// TIA Portal V18 export
// export: Created 2026-06-08T16:52:55.5874896Z, ExportSetting WithDefaults, DisplayName Totally Integrated Automation Portal, DisplayVersion V18, DisplayName TIA Portal Openness, DisplayVersion V18, DisplayName TIA Portal Version Control Interface, DisplayVersion V18, DisplayName STEP 7 Professional, DisplayVersion V18, DisplayName STEP 7 Safety, DisplayVersion V18, DisplayName WinCC Professional, DisplayVersion V18
VAR_GLOBAL   // PLC tag table "Default tag table"
   Start AT %M0.0 : Bool;
   Fan AT %Q0.0 : Bool;
   "Fan Out Delay" AT %MD2 : Time;
   "Element Start" AT %M0.1 : Bool;
   Element AT %Q0.2 : Bool;
   "Element Time Delay" AT %MD6 : Time;
   "Start Up" AT %M0.2 : Bool;
   "Start Up Delay" AT %MD10 : Time;
   Auger AT %Q0.1 : Bool;
   RTD AT %IW96 : Word;
   "RTD 2" AT %IW98 : Word;
   Setpoint AT %MW20 : Word;
   "RTD Real" AT %MD14 : Real;
   "RTD 2 Real" AT %MD22 : Real;
   "Corrected RTD Temp" AT %MD26 : Real;
   "Corrected RTD 2 Temp" AT %MD30 : Real;
   "Auger PID" AT %M0.3 : Bool;
   "Corrected Setpoint" AT %MD34 : Real;
   "Auger Start Up" AT %M0.4 : Bool;
   "Auger Duty Cycle Start" AT %M0.5 : Bool;
   "Auger Duty Cycle" AT %M0.6 : Bool;
   "Auger Duty Cycle Output" AT %M0.7 : Bool;
   "Test Output" AT %M1.0 : Bool;
   "Set Reset" AT %M1.1 : Bool;
   "Error Ack" AT %M1.2 : Bool;
   "Error Ack Button" AT %M1.3 : Bool;
END_VAR
